// TIA Portal V17 export
// export: Created 2025-06-26T07:49:14.6718289Z, ExportSetting WithDefaults, DisplayName Totally Integrated Automation Portal, DisplayVersion V17 Update 8, DisplayName TIA Portal Openness, DisplayVersion V17 Update 8, DisplayName TIA Portal Version Control Interface, DisplayVersion V17, DisplayName STEP 7 Professional, DisplayVersion V17 Update 8, DisplayName STEP 7 Safety, DisplayVersion V17 Update 6, DisplayName WinCC Advanced, DisplayVersion V17 Update 8
FUNCTION_BLOCK "S7_Internal"   // FB1, FBD
TITLE = Exchange data with Process PLC
{ S7_Optimized_Access := 'TRUE' }
VERSION : 0.1
// NOTES:
// 1. Size of CalcValue: 14 bytes
// 2. Max size one GET block can do: 222 bytes
// 3. Max. approx 10 simultaneous GET requests, so broken up into groups
// 4. Only one group is active per cycle. Total update cycle time is (Groups * OB31 cycle time)
// 5. REQ must stay high until the GET has completed (level signal). An edge on REQ will not work.
// 6. When a GET has completed it raises NDR for one cycle. The whole group is complete when all NDRs have been raised. GETs in the same group may not complete in the same cycle, so each NDR is used to SET a bit in xGroup to prevent retriggering while waiting (and thus getting stuck in that group as the NDRs will never go high at the same time). This is actually a sign that the OB cyclic rate is faster than the communication runs (two or more cycles per group) and that it should be increased, but at least it doesn't get stuck.
// 7. More groups can be added by following the model. WARNING: don't play here unless you are prepared for the consequences :-)
// stored: AutoNumber true, IsIECCheckEnabled false, IsRetainMemResEnabled false, MemoryReserve 100, SetENOAutomatically false, UDAEnableTagReadback false
   VAR_INPUT
      bEnable : Bool;   // 1 = do S7 comm, 0 = inhibit
   END_VAR
   VAR
      nGroup : USInt := 1;   // Read group
      xGroup1 : Byte;   // Group 1 read complete status bits
      xGroup2 : Byte;   // Group 2 read complete status bits
      xGroup3 : Byte;   // Group 3 read complete status bits
      xGroup4 : Byte;   // Group 4 read complete status bits
      GET_1 { S7_SetPoint := 'True'} : GET;
      GET_2 { S7_SetPoint := 'True'} : GET;
      GET_3 { S7_SetPoint := 'True'} : GET;
      GET_AI_4 { S7_SetPoint := 'True'} : GET;
      GET_AI_5 { S7_SetPoint := 'True'} : GET;
      GET_AI_6 { S7_SetPoint := 'True'} : GET;
      GET_AI_7 { S7_SetPoint := 'True'} : GET;
      GET_AI_8 { S7_SetPoint := 'True'} : GET;
      PUT_1 { S7_SetPoint := 'True'} : PUT;
      CommCycles { S7_SetPoint := 'True'} : UDInt;
      Group1Timeout : TON_TIME;
      Group2Timeout { S7_SetPoint := 'True'} : TON_TIME;
      Group3Timeout { S7_SetPoint := 'True'} : TON_TIME;
      Group4Timeout { S7_SetPoint := 'True'} : TON_TIME;
      RuntimeMemory { S7_SetPoint := 'True'} : LReal;
      RuntimeElapsed : LReal;   // How long one comm cycle takes
   END_VAR
   VAR_TEMP
      Group1Done : Bool;
      Group2Done : Bool;
      Group3Done : Bool;
      Group4Done : Bool;
   END_VAR
   VAR CONSTANT
      GroupTimeout : Time := T#3s;
   END_VAR
   VAR_TEMP   // added for the SCL form of the ladder/FBD networks
      _w1 : Bool;
   END_VAR
BEGIN

REGION Network 1: Group 1: GET
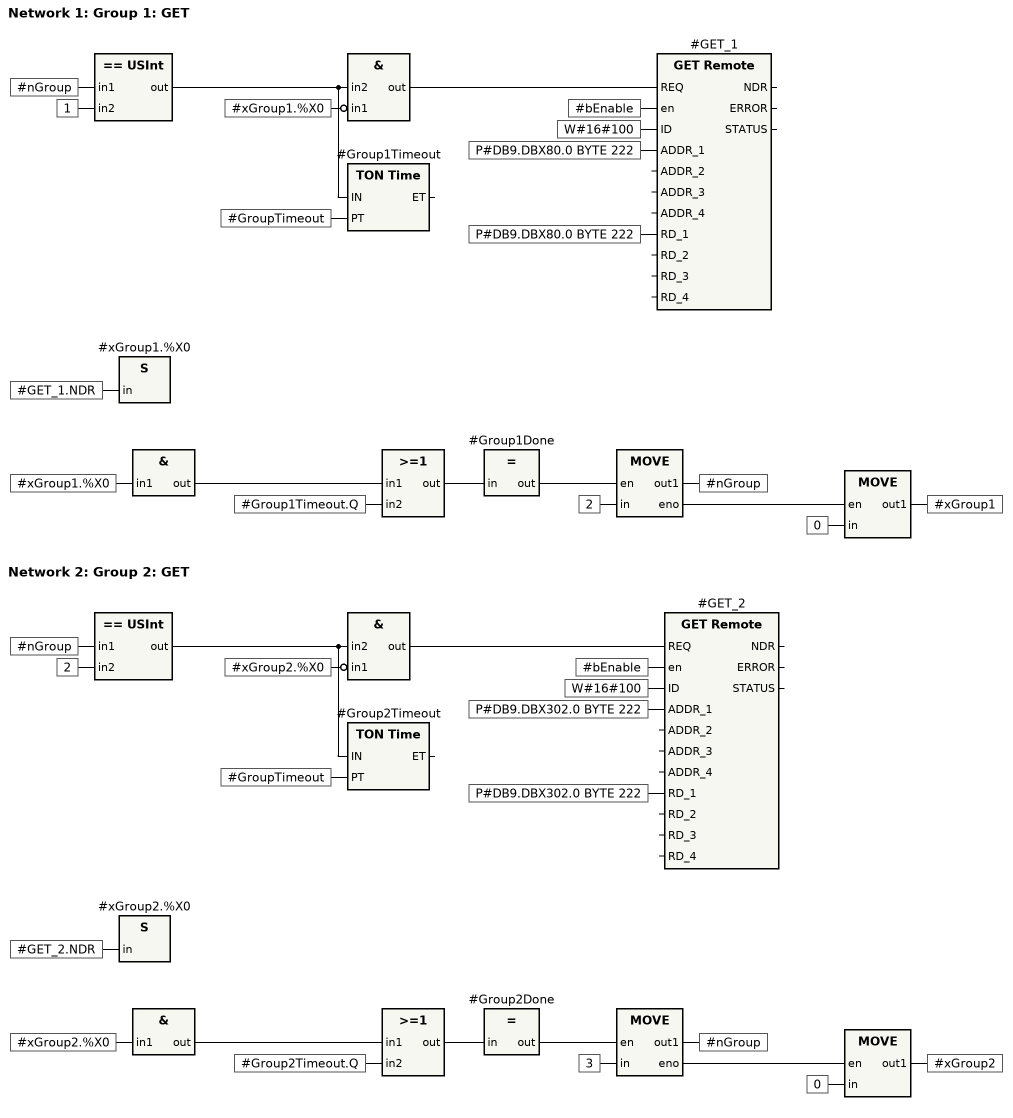
   #_w1 := #nGroup = 1;
   IF #bEnable THEN
       #GET_1(REQ := #_w1 AND NOT #xGroup1.%X0,   // GET
              ID := W#16#100,
              ADDR_1 := P#DB9.DBX80.0 BYTE 222,
              RD_1 := P#DB9.DBX80.0 BYTE 222);
   END_IF;
   #Group1Timeout(IN := #_w1, PT := #GroupTimeout);   // TON
   IF #GET_1.NDR THEN #xGroup1.%X0 := TRUE; END_IF;
   #Group1Done := #xGroup1.%X0 OR #Group1Timeout.Q;
   IF #Group1Done THEN
       #nGroup := 2;
       #xGroup1 := 0;
   END_IF;
END_REGION

REGION Network 2: Group 2: GET
   #_w1 := #nGroup = 2;
   IF #bEnable THEN
       #GET_2(REQ := #_w1 AND NOT #xGroup2.%X0,   // GET
              ID := W#16#100,
              ADDR_1 := P#DB9.DBX302.0 BYTE 222,
              RD_1 := P#DB9.DBX302.0 BYTE 222);
   END_IF;
   #Group2Timeout(IN := #_w1, PT := #GroupTimeout);   // TON
   IF #GET_2.NDR THEN #xGroup2.%X0 := TRUE; END_IF;
   #Group2Done := #xGroup2.%X0 OR #Group2Timeout.Q;
   IF #Group2Done THEN
       #nGroup := 3;
       #xGroup2 := 0;
   END_IF;
END_REGION

REGION Network 3: Group 3: GET
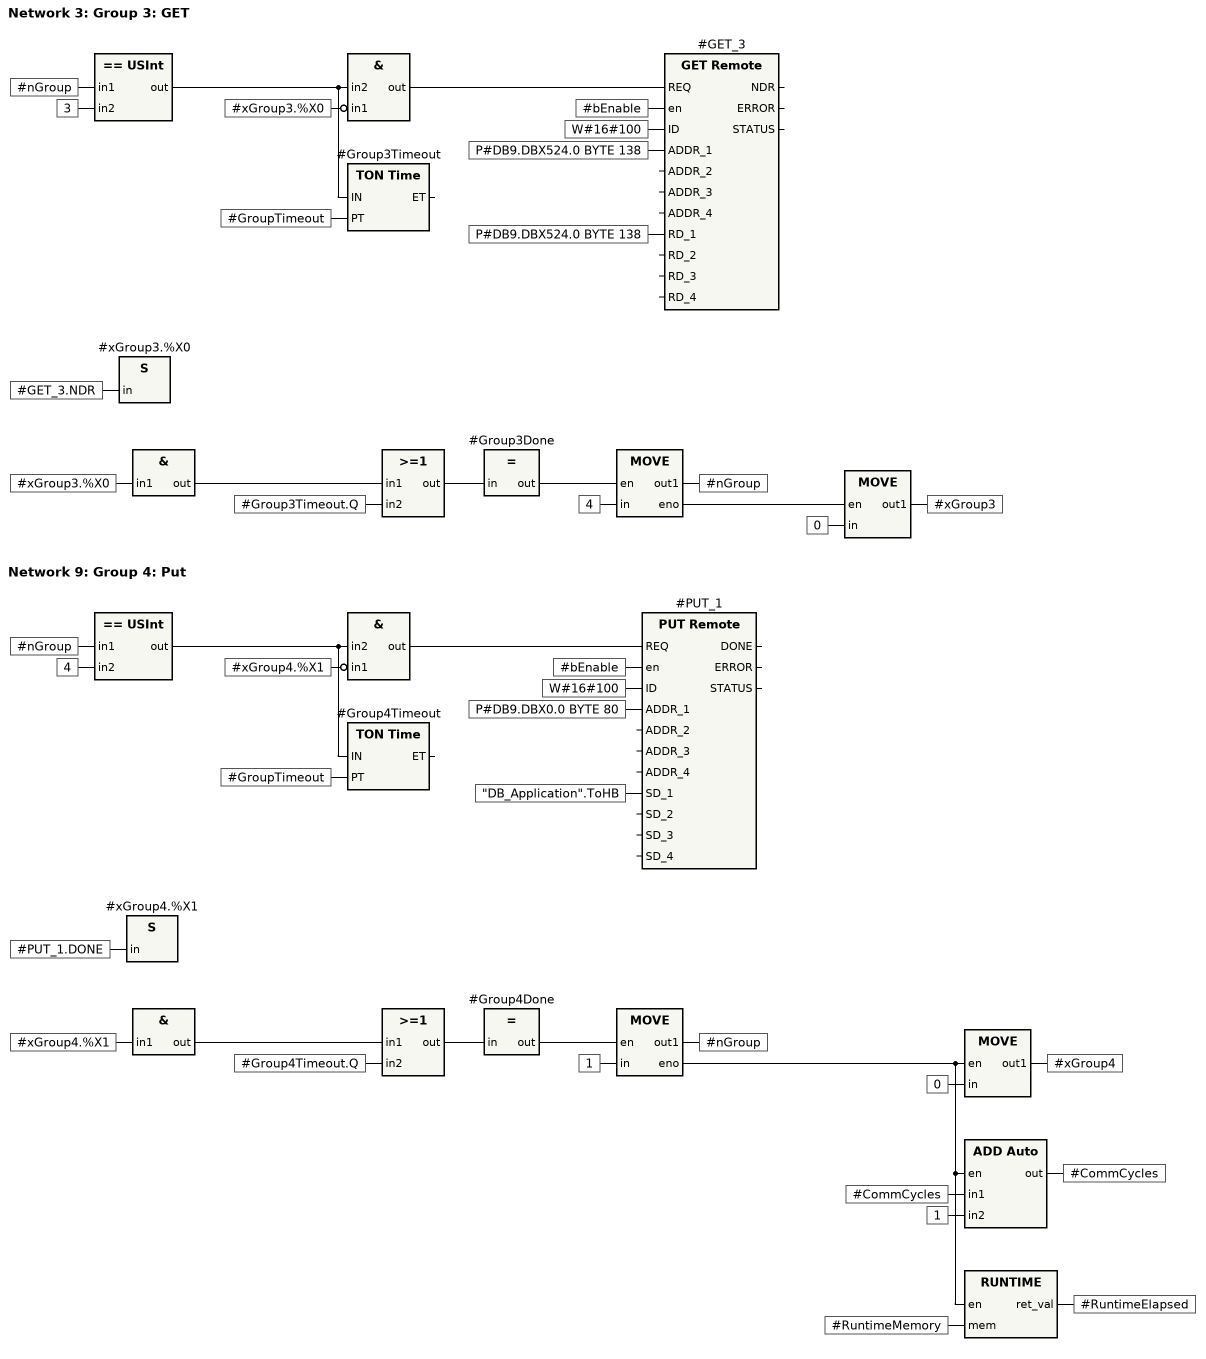
   #_w1 := #nGroup = 3;
   IF #bEnable THEN
       #GET_3(REQ := #_w1 AND NOT #xGroup3.%X0,   // GET
              ID := W#16#100,
              ADDR_1 := P#DB9.DBX524.0 BYTE 138,
              RD_1 := P#DB9.DBX524.0 BYTE 138);
   END_IF;
   #Group3Timeout(IN := #_w1, PT := #GroupTimeout);   // TON
   IF #GET_3.NDR THEN #xGroup3.%X0 := TRUE; END_IF;
   #Group3Done := #xGroup3.%X0 OR #Group3Timeout.Q;
   IF #Group3Done THEN
       #nGroup := 4;
       #xGroup3 := 0;
   END_IF;
END_REGION

REGION Network 4 (SCL): DB_AI
   // Update on new value
   IF #Group3Done = TRUE THEN
       "DB_Heatbooster".AI.HBL_TT_502.fValue := "DB_Application".FromHB.DB_AI.HBL_TT_502;
       "DB_Heatbooster".AI.HBL_PT_503.fValue := "DB_Application".FromHB.DB_AI.HBL_PT_503;
       "DB_Heatbooster".AI.HBL_TT_504.fValue := "DB_Application".FromHB.DB_AI.HBL_TT_504;
       "DB_Heatbooster".AI.HBL_LT_510.fValue := "DB_Application".FromHB.DB_AI.HBL_LT_510;
       "DB_Heatbooster".AI.HBL_PT_511.fValue := "DB_Application".FromHB.DB_AI.HBL_PT_511;
       "DB_Heatbooster".AI.HBL_TT_512.fValue := "DB_Application".FromHB.DB_AI.HBL_TT_512;
       "DB_Heatbooster".AI.HBL_TT_516.fValue := "DB_Application".FromHB.DB_AI.HBL_TT_516;
       "DB_Heatbooster".AI.HBL_PT_517.fValue := "DB_Application".FromHB.DB_AI.HBL_PT_517;
       "DB_Heatbooster".AI.HBL_TT_518.fValue := "DB_Application".FromHB.DB_AI.HBL_TT_518;
       "DB_Heatbooster".AI.HBL_PT_519.fValue := "DB_Application".FromHB.DB_AI.HBL_PT_519;
       "DB_Heatbooster".AI.HBL_FT_520.fValue := "DB_Application".FromHB.DB_AI.HBL_FT_520;
       "DB_Heatbooster".AI.HBL_TT_530.fValue := "DB_Application".FromHB.DB_AI.HBL_TT_530;
       "DB_Heatbooster".AI.HBL_PT_531.fValue := "DB_Application".FromHB.DB_AI.HBL_PT_531;
       "DB_Heatbooster".AI.HBL_TT_532.fValue := "DB_Application".FromHB.DB_AI.HBL_TT_532;
       "DB_Heatbooster".AI.HBL_TT_533.fValue := "DB_Application".FromHB.DB_AI.HBL_TT_533;
       "DB_Heatbooster".AI.HBL_PT_534.fValue := "DB_Application".FromHB.DB_AI.HBL_PT_534;
       "DB_Heatbooster".AI.HBL_AT_535.fValue := "DB_Application".FromHB.DB_AI.HBL_AT_535;
       "DB_Heatbooster".AI.HBL_TT_540.fValue := "DB_Application".FromHB.DB_AI.HBL_TT_540;
       "DB_Heatbooster".AI.HBL_PT_541.fValue := "DB_Application".FromHB.DB_AI.HBL_PT_541;
       "DB_Heatbooster".AI.HBL_TT_542.fValue := "DB_Application".FromHB.DB_AI.HBL_TT_542;
       "DB_Heatbooster".AI.HBL_TT_543.fValue := "DB_Application".FromHB.DB_AI.HBL_TT_543;
       "DB_Heatbooster".AI.HBL_PT_544.fValue := "DB_Application".FromHB.DB_AI.HBL_PT_544;
       "DB_Heatbooster".AI.HBL_AT_545.fValue := "DB_Application".FromHB.DB_AI.HBL_AT_545;
       "DB_Heatbooster".AI.HBL_TT_546.fValue := "DB_Application".FromHB.DB_AI.HBL_TT_546;
       "DB_Heatbooster".AI.HBL_PT_547.fValue := "DB_Application".FromHB.DB_AI.HBL_PT_547;
       "DB_Heatbooster".AI.HBL_TT_571.fValue := "DB_Application".FromHB.DB_AI.HBL_TT_571;
       "DB_Heatbooster".AI.HBL_PT_572.fValue := "DB_Application".FromHB.DB_AI.HBL_PT_572;
       "DB_Heatbooster".AI.HBL_TT_573.fValue := "DB_Application".FromHB.DB_AI.HBL_TT_573;
       "DB_Heatbooster".AI.HBL_LT_610.fValue := "DB_Application".FromHB.DB_AI.HBL_LT_610;
       "DB_Heatbooster".AI.HBL_TT_611.fValue := "DB_Application".FromHB.DB_AI.HBL_TT_611;
       "DB_Heatbooster".AI.HBL_PT_612.fValue := "DB_Application".FromHB.DB_AI.HBL_PT_612;
       "DB_Heatbooster".AI.HBL_CT_615.fValue := "DB_Application".FromHB.DB_AI.HBL_CT_615;
       "DB_Heatbooster".AI.HBL_PT_618.fValue := "DB_Application".FromHB.DB_AI.HBL_PT_618;
       "DB_Heatbooster".AI.HBL_PT_635.fValue := "DB_Application".FromHB.DB_AI.HBL_PT_635;
       "DB_Heatbooster".AI.HBL_PT_636.fValue := "DB_Application".FromHB.DB_AI.HBL_PT_636;
       "DB_Heatbooster".AI.HBL_LT_650.fValue := "DB_Application".FromHB.DB_AI.HBL_LT_650;
       "DB_Heatbooster".AI.HBL_PT_651.fValue := "DB_Application".FromHB.DB_AI.HBL_PT_651;
       "DB_Heatbooster".AI.HBL_PT_701.fValue := "DB_Application".FromHB.DB_AI.HBL_PT_701;
       "DB_Heatbooster".AI.HBL_PT_702.fValue := "DB_Application".FromHB.DB_AI.HBL_PT_702;
       "DB_Heatbooster".AI.HBL_PT_703.fValue := "DB_Application".FromHB.DB_AI.HBL_PT_703;
       "DB_Heatbooster".AI.CPC_LT_870.fValue := "DB_Application".FromHB.DB_AI.CPC_LT_870;
       "DB_Heatbooster".AI.CPC_TT_871.fValue := "DB_Application".FromHB.DB_AI.CPC_TT_871;
       "DB_Heatbooster".AI.CPC_PT_872.fValue := "DB_Application".FromHB.DB_AI.CPC_PT_872;
       "DB_Heatbooster".AI.CPC_PT_862.fValue := "DB_Application".FromHB.DB_AI.CPC_PT_862;
       "DB_Heatbooster".AI.HBL_TT_901.fValue := "DB_Application".FromHB.DB_AI.HBL_TT_901;
       "DB_Heatbooster".AI.HBL_PT_902.fValue := "DB_Application".FromHB.DB_AI.HBL_PT_902;

       "DB_Heatbooster".AI.HBL_TT_03.fValue := "DB_Application".FromHB.DB_AI.HBL_TT_03;
       "DB_Heatbooster".AI.HBL_TT_16.fValue := "DB_Application".FromHB.DB_AI.HBL_TT_16;
       "DB_Heatbooster".AI.HBL_TT_17.fValue := "DB_Application".FromHB.DB_AI.HBL_TT_17;
       "DB_Heatbooster".AI.HBL_TT_18.fValue := "DB_Application".FromHB.DB_AI.HBL_TT_18;
       "DB_Heatbooster".AI.HBL_TT_20.fValue := "DB_Application".FromHB.DB_AI.HBL_TT_20;
       "DB_Heatbooster".AI.HBL_TT_21.fValue := "DB_Application".FromHB.DB_AI.HBL_TT_21;
       "DB_Heatbooster".AI.HBL_TT_22.fValue := "DB_Application".FromHB.DB_AI.HBL_TT_22;
       "DB_Heatbooster".AI.HBL_TT_23.fValue := "DB_Application".FromHB.DB_AI.HBL_TT_23;
       "DB_Heatbooster".AI.HBL_TT_24.fValue := "DB_Application".FromHB.DB_AI.HBL_TT_24;
       "DB_Heatbooster".AI.HBL_TT_25.fValue := "DB_Application".FromHB.DB_AI.HBL_TT_25;
       "DB_Heatbooster".AI.HBL_TT_26.fValue := "DB_Application".FromHB.DB_AI.HBL_TT_26;
       "DB_Heatbooster".AI.HBL_TT_27.fValue := "DB_Application".FromHB.DB_AI.HBL_TT_27;
       "DB_Heatbooster".AI.HBL_PT_05.fValue := "DB_Application".FromHB.DB_AI.HBL_PT_05;
       "DB_Heatbooster".AI.HBL_PT_06.fValue := "DB_Application".FromHB.DB_AI.HBL_PT_06;
       "DB_Heatbooster".AI.HBL_PT_17.fValue := "DB_Application".FromHB.DB_AI.HBL_PT_17;
       "DB_Heatbooster".AI.HBL_CT_01.fValue := "DB_Application".FromHB.DB_AI.HBL_CT_01;
       "DB_Heatbooster".AI.HBL_CT_03.fValue := "DB_Application".FromHB.DB_AI.HBL_CT_03;

       "DB_Heatbooster".AI.SSC_TT_01.fValue := "DB_Application".FromHB.DB_AI.SSC_TT_01;
       "DB_Heatbooster".AI.SSC_TT_02.fValue := "DB_Application".FromHB.DB_AI.SSC_TT_02;
       "DB_Heatbooster".AI.SSC_TT_03.fValue := "DB_Application".FromHB.DB_AI.SSC_TT_03;
       "DB_Heatbooster".AI.SSC_TT_04.fValue := "DB_Application".FromHB.DB_AI.SSC_TT_04;
       "DB_Heatbooster".AI.SSC_PIT_01.fValue := "DB_Application".FromHB.DB_AI.SSC_PIT_01;
       "DB_Heatbooster".AI.SSC_PDT_01.fValue := "DB_Application".FromHB.DB_AI.SSC_PDT_01;
       "DB_Heatbooster".AI.SSC_LT_01.fValue := "DB_Application".FromHB.DB_AI.SSC_LT_01;
   END_IF;
END_REGION

REGION Network 5 (SCL): DB_Calc
   IF #Group3Done = TRUE THEN
       "DB_Heatbooster".Calc.Compressor.CrankcaseSaturationTemperature.fValue                      := "DB_Application".FromHB.DB_Calc.Compressor_CrankcaseSaturationTemperature;
       "DB_Heatbooster".Calc.Compressor.CrankcaseSuperheat.fValue                                  := "DB_Application".FromHB.DB_Calc.Compressor_CrankcaseSuperheat;
       "DB_Heatbooster".Calc.Compressor.VolumetricEfficiency.fValue                                := "DB_Application".FromHB.DB_Calc.Compressor_VolumetricEfficiency;
       "DB_Heatbooster".Calc.Compressor.IsentropicEfficiency.fValue                                := "DB_Application".FromHB.DB_Calc.Compressor_IsentropicEfficiency;
       "DB_Heatbooster".Calc.Compressor.Massflow.fValue                                            := "DB_Application".FromHB.DB_Calc.Compressor_Massflow;

       "DB_Heatbooster".Calc.HeatSink.DeltaT.fValue                                                := "DB_Application".FromHB.DB_Calc.Heatsink_DeltaT;         
       "DB_Heatbooster".Calc.HeatSink.Pinch.fValue                                                 := "DB_Application".FromHB.DB_Calc.Heatsink_Pinch;
       "DB_Heatbooster".Calc.HeatSink.HeatRate.fValue                                              := "DB_Application".FromHB.DB_Calc.Heatsink_Heatrate;              
       "DB_Heatbooster".Calc.HeatSink.DeltaP.fValue                                                := "DB_Application".FromHB.DB_Calc.Heatsink_DeltaP;
       "DB_Heatbooster".Calc.HeatSink.Massflow.fValue                                              := "DB_Application".FromHB.DB_Calc.Heatsink_Massflow;

       "DB_Heatbooster".Calc.HeatSource.DeltaT.fValue                                              := "DB_Application".FromHB.DB_Calc.Heatsource_DeltaT;           
       "DB_Heatbooster".Calc.HeatSource.Pinch.fValue                                               := "DB_Application".FromHB.DB_Calc.Heatsource_Pinch;
       "DB_Heatbooster".Calc.HeatSource.HeatRate.fValue                                            := "DB_Application".FromHB.DB_Calc.Heatsource_Heatrate;
       "DB_Heatbooster".Calc.HeatSource.DeltaP.fValue                                              := "DB_Application".FromHB.DB_Calc.Heatsource_DeltaP;
       "DB_Heatbooster".Calc.HeatSource.Massflow.fValue                                            := "DB_Application".FromHB.DB_Calc.Heatsource_Massflow;
       "DB_Heatbooster".Calc.HeatSource.TemperatureRateOfChange.fValue                             := "DB_Application".FromHB.DB_Calc.Heatsource_TemperatureRateOfChange;

       "DB_Heatbooster".Calc.HighPressPart.CompressorSaturationTemperature.fValue                  := "DB_Application".FromHB.DB_Calc.HighPressPart_CompressorSaturationTemperature;
       "DB_Heatbooster".Calc.HighPressPart.CompressorSuperheat.fValue                              := "DB_Application".FromHB.DB_Calc.HighPressPart_CompressorSuperheat;
       "DB_Heatbooster".Calc.HighPressPart.CondenserSaturationTemperature.fValue                   := "DB_Application".FromHB.DB_Calc.HighPressPart_CondenserSaturationTemperature;
       "DB_Heatbooster".Calc.HighPressPart.CondenserSubcooling.fValue                              := "DB_Application".FromHB.DB_Calc.HighPressPart_CondenserSubcooling;
       "DB_Heatbooster".Calc.HighPressPart.ExpansionValveSubcooling.fValue                         := "DB_Application".FromHB.DB_Calc.HighPressPart_ExpansionValveSubcooling;
       "DB_Heatbooster".Calc.HighPressPart.CondenserDeltaP.fValue                                  := "DB_Application".FromHB.DB_Calc.HighPressPart_CondenserDeltaP;

       "DB_Heatbooster".Calc.LowPressPart.EvaporatorSuperheat.fValue                               := "DB_Application".FromHB.DB_Calc.LowPressPart_EvaporatorSuperheat;
       "DB_Heatbooster".Calc.LowPressPart.CompressorSuperheat.fValue                               := "DB_Application".FromHB.DB_Calc.LowPressPart_CompressorSuperheat;
       "DB_Heatbooster".Calc.LowPressPart.EvaporatorSaturationTemperature.fValue                   := "DB_Application".FromHB.DB_Calc.LowPressPart_EvaporatorSaturationTemperature;
       "DB_Heatbooster".Calc.LowPressPart.CompressorSaturationTemperature.fValue                   := "DB_Application".FromHB.DB_Calc.LowPressPart_CompressorSaturationTemperature;

       "DB_Heatbooster".Calc.System.Quality.fValue                                                 := "DB_Application".FromHB.DB_Calc.System_Quality;
       "DB_Heatbooster".Calc.System.COP.fValue                                                     := "DB_Application".FromHB.DB_Calc.System_COP;
       "DB_Heatbooster".Calc.System.ElectricalPower.fValue                                         := "DB_Application".FromHB.DB_Calc.System_ElectricalPower;
       "DB_Heatbooster".Calc.System.TemperatureLift.fValue                                         := "DB_Application".FromHB.DB_Calc.System_TemperatureLift;      
       "DB_Heatbooster".Calc.System.MotorEfficiency.fValue                                         := "DB_Application".FromHB.DB_Calc.System_MotorEfficiency;                      
       "DB_Heatbooster".Calc.System.FMEP.fValue                                                    := "DB_Application".FromHB.DB_Calc.System_FMEP;                      

       "DB_Heatbooster".Calc.Auxiliary.ShaftSealDeltaT.fValue                                      := "DB_Application".FromHB.DB_Calc.Aux_ShaftSealDeltaT;
       "DB_Heatbooster".Calc.Auxiliary.CPCPumpDeltaP.fValue                                        := "DB_Application".FromHB.DB_Calc.Aux_CPCPumpDeltaP;

       "DB_Heatbooster".Calc.Misc.EvaporatorDischargePressureMean.fValue                           := "DB_Application".FromHB.DB_Calc.Misc_EvaporatorDischargePressureMean;
       "DB_Heatbooster".Calc.Misc.EvaporatorDischargeTemperatureMin.fValue                         := "DB_Application".FromHB.DB_Calc.Misc_EvaporatorDischargeTemperatureMin;
       "DB_Heatbooster".Calc.Misc.EvaporatorDischargeTemperatureMean.fValue                        := "DB_Application".FromHB.DB_Calc.Misc_EvaporatorDischargeTemperatureMean;
       "DB_Heatbooster".Calc.Misc.OilFilterDeltaP.fValue                                           := "DB_Application".FromHB.DB_Calc.Misc_OilFilterDeltaP;
   END_IF;
END_REGION

REGION Network 6 (SCL): DB_InverterDrives & DB_Valves
   IF #Group3Done = TRUE THEN
       "DB_Heatbooster".Inverter.HBL_SC_01_A1.fValue    := "DB_Application".FromHB.DB_InverterDrives.HBL_SC_01_A1;  
       "DB_Heatbooster".Inverter.HBL_SC_01_A2.fValue    := "DB_Application".FromHB.DB_InverterDrives.HBL_SC_01_A2;  
       "DB_Heatbooster".Inverter.HBL_SC_01_A3.fValue    := "DB_Application".FromHB.DB_InverterDrives.HBL_SC_01_A3;  
       "DB_Heatbooster".Inverter.HBL_SC_02_A1.fValue    := "DB_Application".FromHB.DB_InverterDrives.HBL_SC_02_A1;  
       "DB_Heatbooster".Inverter.HBL_SC_02_A2.fValue    := "DB_Application".FromHB.DB_InverterDrives.HBL_SC_02_A2;  
       "DB_Heatbooster".Inverter.HBL_SC_02_A3.fValue    := "DB_Application".FromHB.DB_InverterDrives.HBL_SC_02_A3;  
       "DB_Heatbooster".Inverter.HBL_SC_10_A1.fValue    := "DB_Application".FromHB.DB_InverterDrives.HBL_SC_10_A1;  
       "DB_Heatbooster".Inverter.HBL_SC_10_A2.fValue    := "DB_Application".FromHB.DB_InverterDrives.HBL_SC_10_A2;  
       "DB_Heatbooster".Inverter.HBL_SC_10_A3.fValue    := "DB_Application".FromHB.DB_InverterDrives.HBL_SC_10_A3;
       "DB_Heatbooster".Inverter.HBL_SC_03_A1.fValue   := "DB_Application".FromHB.DB_InverterDrives.HBL_SC_03_A1;
       "DB_Heatbooster".Inverter.HBL_SC_03_A2.fValue   := "DB_Application".FromHB.DB_InverterDrives.HBL_SC_03_A2;
       "DB_Heatbooster".Inverter.HBL_SC_03_A3.fValue   := "DB_Application".FromHB.DB_InverterDrives.HBL_SC_03_A3;


       "DB_Heatbooster".Valve.HBL_HCV_576_A1.fValue          := "DB_Application".FromHB.DB_Valves.HBL_HCV_576_A1;  
       "DB_Heatbooster".Valve.HBL_HCV_578_A1.fValue          := "DB_Application".FromHB.DB_Valves.HBL_HCV_578_A1;
       "DB_Heatbooster".Valve.HBL_HCV_577_A1.fValue          := "DB_Application".FromHB.DB_Valves.HBL_HCV_577_A1;
       "DB_Heatbooster".Valve.HBL_HCV_579_A1.fValue          := "DB_Application".FromHB.DB_Valves.HBL_HCV_579_A1;
       "DB_Heatbooster".Valve.HBL_HCV_515_A1.fValue          := "DB_Application".FromHB.DB_Valves.HBL_HCV_515_A1;
       "DB_Heatbooster".Valve.HBL_HCV_575_A1.fValue          := "DB_Application".FromHB.DB_Valves.HBL_HCV_575_A1;
       "DB_Heatbooster".Valve.HBL_HCV_616_A1.fValue          := "DB_Application".FromHB.DB_Valves.HBL_HCV_616_A1;
       "DB_Heatbooster".Valve.HBL_HCV_700_A1.fValue          := "DB_Application".FromHB.DB_Valves.HBL_HCV_700_A1;
       "DB_Heatbooster".Valve.HBL_HCV_514_A1.fValue := "DB_Application".FromHB.DB_Valves.HBL_HCV_514_A1;
       "DB_Heatbooster".Valve.HBL_HCV_548_A1.fValue := "DB_Application".FromHB.DB_Valves.HBL_HCV_548_A1;


   END_IF;
END_REGION

REGION Network 7 (SCL): DB_DO
   IF #Group3Done = TRUE THEN
       "DB_DO".HBL_EC_01 := "DB_Application".FromHB.OilHeatersGroup1;
       "DB_DO".HBL_EC_02 := "DB_Application".FromHB.OilHeatersGroup2;
       "DB_DO".HBL_HV_630 := "DB_Application".FromHB.HBL_HV_630;
       "DB_DO".HBL_HV_631 := "DB_Application".FromHB.HBL_HV_631;
       "DB_DO".HBL_HV_860 := "DB_Application".FromHB.HBL_HV_860;
       "DB_DO".HBL_HV_861 := "DB_Application".FromHB.HBL_HV_861;
       "DB_DO".SSC_P_01  := "DB_Application".FromHB.SSC_P_01;
       "DB_DO".SSC_F_01 := "DB_Application".FromHB.SSC_F_01;
       "DB_DO".SSC_P_02  := "DB_Application".FromHB.SSC_P_02;
       "DB_DO".CPC_P_01  := "DB_Application".FromHB.CPC_P_01;
       "DB_DO".HBL_LSH_62 := "DB_Application".FromHB.HBL_LSH_62;
       "DB_DO".HBL_LSL_63 := "DB_Application".FromHB.HBL_LSL_63;
       "DB_DO".HBL_LSH_64 := "DB_Application".FromHB.HBL_LSH_64;
       "DB_DO".HBL_LSL_864 := "DB_Application".FromHB.HBL_LSL_864;
       "DB_DO".HBL_LS_632 := "DB_Application".FromHB.HBL_LS_632;
       "DB_DO".HBL_LS_633 := "DB_Application".FromHB.HBL_LS_633;

   END_IF;
END_REGION

REGION Network 8 (SCL): Mapping to HB PLC
   // Things that could/should be directly connected to the Heatbooster, but are not
   "DB_Application".ToHB.HBL_HCV_514_A1 := "DB_TestSupport".Valve.TSA_HCV_322_A1.fValue;
   "DB_Application".ToHB.HBL_HCV_548_A1 := "DB_TestSupport".Valve.TSA_HCV_370_A1.fValue;
   "DB_Application".ToHB.HBL_TT_546 := "DB_TestSupport".AI.TSA_TT_356.fValue;
   "DB_Application".ToHB.HBL_PT_547 := "DB_TestSupport".AI.TSA_PT_374.fValue;
   "DB_Application".ToHB.HBL_HCV_515_A1 := 0.0; // no such valve installed 
   "DB_Application".ToHB.HBL_TT_901 := "DB_TestSupport".AI.TSA_TT_301.fValue;
   "DB_Application".ToHB.HBL_PT_902 := "DB_TestSupport".AI.TSA_PT_300.fValue;
   "DB_Application".ToHB.HBL_TT_512 := "DB_TestSupport".AI.TSA_TT_320.fValue;
   "DB_Application".ToHB.HBL_PT_511 := "DB_TestSupport".AI.TSA_PT_321.fValue;
   "DB_Application".ToHB.HBL_PT_519 := "DB_TestSupport".AI.TSA_PT_323.fValue;
   "DB_Application".ToHB.HBL_TT_518 := "DB_TestSupport".AI.TSA_TT_324.fValue;
   "DB_Application".ToHB.LivenessCounter := UDINT_TO_UINT(#CommCycles);
END_REGION

REGION Network 9: Group 4: Put
   // no SCL statement known for Runtime: written as a call
   #_w1 := #nGroup = 4;
   IF #bEnable THEN
       #PUT_1(REQ := #_w1 AND NOT #xGroup4.%X1,   // PUT
              ID := W#16#100,
              ADDR_1 := P#DB9.DBX0.0 BYTE 80,
              SD_1 := "DB_Application".ToHB);
   END_IF;
   #Group4Timeout(IN := #_w1, PT := #GroupTimeout);   // TON
   IF #PUT_1.DONE THEN #xGroup4.%X1 := TRUE; END_IF;
   #Group4Done := #xGroup4.%X1 OR #Group4Timeout.Q;
   IF #Group4Done THEN
       #nGroup := 1;
       #xGroup4 := 0;
       #CommCycles := #CommCycles + 1;
       #RuntimeElapsed := Runtime(mem := #RuntimeMemory);
   END_IF;
END_REGION
END_FUNCTION_BLOCK
